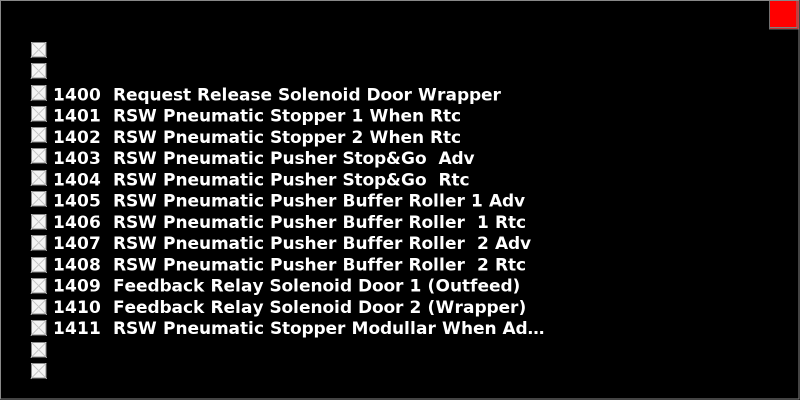
VISUALIZATION P2_DI5  // 800x400, background image 
    ImageSwitcher (31,42 15x15), variable: InputOutput_GVL.Digital_Input[65], behaviour: TOGGLE
    Label (50,16 625x391), "1400 Request Release Solenoid Door Wrapper 1401 RSW Pneumatic Stopper 1 When Rtc 1402 RSW Pneumatic Stopper 2 When Rtc 1403 RSW Pneumatic Pusher Stop&Go Adv 1404 RSW Pneumatic Pusher Stop&Go Rtc 1405 RSW Pneumatic Pusher Buffer Roller 1 Adv 1406 RSW Pneumatic Pusher Buffer Roller 1 Rtc 1407 RSW Pneumatic Pusher Buffer Roller 2 Adv 1408 RSW Pneumatic Pusher Buffer Roller 2 Rtc 1409 Feedback Relay Solenoid Door 1 (Outfeed) 1410 Feedback Relay Solenoid Door 2 (Wrapper) 1411 RSW Pneumatic Stopper Modullar When Adv 1412 RSW Pneumatic Stopper Modullar When Rtc 1413 1414 Interlock Feedback Pallet Ready at Infeed Dispenser 1415 Interlock Feedback Pallet Ready at Unloading"
    ImageSwitcher (31,63 15x15), variable: InputOutput_GVL.Digital_Input[66], behaviour: TOGGLE
    ImageSwitcher (31,85 15x15), variable: InputOutput_GVL.Digital_Input[67], behaviour: TOGGLE
    ImageSwitcher (31,106 15x15), variable: InputOutput_GVL.Digital_Input[68], behaviour: TOGGLE
    ImageSwitcher (31,127 15x15), variable: InputOutput_GVL.Digital_Input[69], behaviour: TOGGLE
    ImageSwitcher (31,148 15x15), variable: InputOutput_GVL.Digital_Input[70], behaviour: TOGGLE
    ImageSwitcher (31,170 15x15), variable: InputOutput_GVL.Digital_Input[71], behaviour: TOGGLE
    ImageSwitcher (31,191 15x15), variable: InputOutput_GVL.Digital_Input[72], behaviour: TOGGLE
    ImageSwitcher (31,214 15x15), variable: InputOutput_GVL.Digital_Input[73], behaviour: TOGGLE
    ImageSwitcher (31,235 15x15), variable: InputOutput_GVL.Digital_Input[74], behaviour: TOGGLE
    ImageSwitcher (31,257 15x15), variable: InputOutput_GVL.Digital_Input[75], behaviour: TOGGLE
    ImageSwitcher (31,278 15x15), variable: InputOutput_GVL.Digital_Input[76], behaviour: TOGGLE
    ImageSwitcher (31,299 15x15), variable: InputOutput_GVL.Digital_Input[77], behaviour: TOGGLE
    ImageSwitcher (31,320 15x15), variable: InputOutput_GVL.Digital_Input[78], behaviour: TOGGLE
    ImageSwitcher (31,342 15x15), variable: InputOutput_GVL.Digital_Input[79], behaviour: TOGGLE
    ImageSwitcher (31,363 15x15), variable: InputOutput_GVL.Digital_Input[80], behaviour: TOGGLE
    Button (769,-1 30x30), image: VisuSymbols.Symbols.Wrong
        OnMouseClick: CloseDialog Dialog=P2_DI5, Result=OK, NumpadKeypadSet=True
END_VISUALIZATION

(* stored: Version 1.1.0.1, ProductVersion 3.1.4024.12
   Visu P2_DI5: Id {1b54dfea-77d6-4ecb-a921-ba98a6f40068} *)
